{attribute 'qualified_only'}
VAR_GLOBAL
	bStart : BOOL;
	bStop : BOOL;
	bTopSwitch : BOOL;
	bManual : BOOL;
	bOn : BOOL;
<<<<<<< HEAD
    eMode : E_modes;
	eStatus : E_Status;
	fJoystickX : LREAL;
	fJoystickY : LREAL;
	bError : BOOL := FALSE;
=======
	eModeSwitch : E_Modes;
>>>>>>> parent of 03fe425 (HMI status ferdig)
END_VAR

(* stored: Version 1.1.0.1, ProductVersion 3.1.4024.12
   GVL task1: Id {94ceed5f-9cf7-441b-a5a5-289e85e116de} *)
